(* CoDeSys 2.3.5.6 project: szlendak_02.pro *)
(* Libraries: Standard.lib 31.10.14 11:17:58, SYSLIBCALLBACK.LIB 31.10.14 11:17:58 *)

(* PLC configuration (modules and I/O channels)
Configuration EC4P-200 [Root] node -1, in %IB0 out %QB0 {EC4P_RestartPwrOn = WARMSTART; EC4P_MaxCycleTime = 20; EC4P_Com1BaudRate = 38400; EC4P_CAN1BaudRate = 125KBaud; EC4P_RoutingId = 127; EC4P_EasyNetId = 1; EC4P_EasyNetCfg = 0; EC4P_EasyNetCycleTime = 50; EC4P_RoutingChannel = CAN1; EC4P_IPFlags = 0; EC4P_IPAddress = 0; EC4P_SubNetMask = 0; EC4P_DefaultGateway = 0; EC4P_SummerWinterFlags = 0; EC4P_SummerWinterRule1 = 0; EC4P_SummerWinterRule2 = 0}
  Local I/O [EC4P_LocalIO] node 0, in %IB0 out %QB0 {EC4P_LocalInt = 0}
    I1 AT %IX0.0 [LocalBitInput] Input I1
    I2 AT %IX0.1 [LocalBitInput] Input I2
    I3 AT %IX0.2 [LocalBitInput] Input I3
    I4 AT %IX0.3 [LocalBitInput] Input I4
    I5 AT %IX0.4 [LocalBitInput] Input I5
    I6 AT %IX0.5 [LocalBitInput] Input I6
    I7 AT %IX0.6 [LocalBitInput] Input I7
    I8 AT %IX0.7 [LocalBitInput] Input I8
    I9 AT %IX1.0 [LocalBitInput] Input I9
    I10 AT %IX1.1 [LocalBitInput] Input I10
    I11 AT %IX1.2 [LocalBitInput] Input I11
    I12 AT %IX1.3 [LocalBitInput] Input I12
    I13 AT %IX1.4 [LocalDiagInput] Diagnostic Input I13
    I14 AT %IX1.5 [LocalDiagInput] Diagnostic Input I14
    I15 AT %IX1.6 [LocalDiagInput] Diagnostic Input I15
    I16 AT %IX1.7 [LocalDiagInput] Diagnostic Input I16
    I7_Analog AT %IW2 [LocalAnalogIn] Input I7, 10Bit, 0-10VDC
    I8_Analog AT %IW4 [LocalAnalogIn] Input I8, 10Bit, 0-10VDC
    I11_Analog AT %IW6 [LocalAnalogIn] Input I11, 10Bit, 0-10VDC
    I12_Analog AT %IW8 [LocalAnalogIn] Input I12, 10Bit, 0-10VDC
    Transistor Outputs [EC4P_TOutputs] node 0, in %IB10 out %QB0
      Q1 AT %QX0.0 [LocalBitOutput] Transistor-Output Q1
      Q2 AT %QX0.1 [LocalBitOutput] Transistor-Output Q2
      Q3 AT %QX0.2 [LocalBitOutput] Transistor-Output Q3
      Q4 AT %QX0.3 [LocalBitOutput] Transistor-Output Q4
      Q5 AT %QX0.4 [LocalBitOutput] Transistor-Output Q5
      Q6 AT %QX0.5 [LocalBitOutput] Transistor-Output Q6
      Q7 AT %QX0.6 [LocalBitOutput] Transistor-Output Q7
      Q8 AT %QX0.7 [LocalBitOutput] Transistor-Output Q8
    No Analog Output [EC4P_NoAnalogOutput] node 1, in %IB10 out %QB1
    No Keys [EC4P_NoKeys] node 2, in %IB10 out %QB1
    No Counter [EC4P_NoCounter] node 3, in %IB10 out %QB1
  Extension [EC4P_Extension] node 1, in %IB10 out %QB1
    No Extension [EC4P_NoExtension] node 0, in %IB10 out %QB1
*)

(* Global variable list: Zmienne_globalne *)
VAR_GLOBAL
	K1: BOOL;
	K2: BOOL;
	K3: BOOL;
	f2: BOOL;
	g2: BOOL;
END_VAR

(* POU PLC_PRG, LD *)
PROGRAM PLC_PRG
VAR
	T1: TON;
	T2: TP;
	T4: F_TRIG;
	T3: TP;
	T5: TP;
	T6: F_TRIG;
	T7: TON;
	T8: TP;
	T9: F_TRIG;
	T10: TP;
	T11: F_TRIG;
	T12: TP;
	T13: TP;
	T14: TP;
	T15: TON;
	T16: TP;
	T17: TON;
	x1: BOOL;
	x2: BOOL;
	r1: R_TRIG;
	to1: TOF;
	y1: BOOL;
	r2: F_TRIG;
	to2: TOF;
	y2: BOOL;
	f4: BOOL;
	f3: BOOL;
	f1: BOOL;
	g1: BOOL;
	f6: BOOL;
	f7: BOOL;
	f8: BOOL;
	g3: BOOL;
	g4: BOOL;
END_VAR
VAR_INPUT
	f5: BOOL;
END_VAR
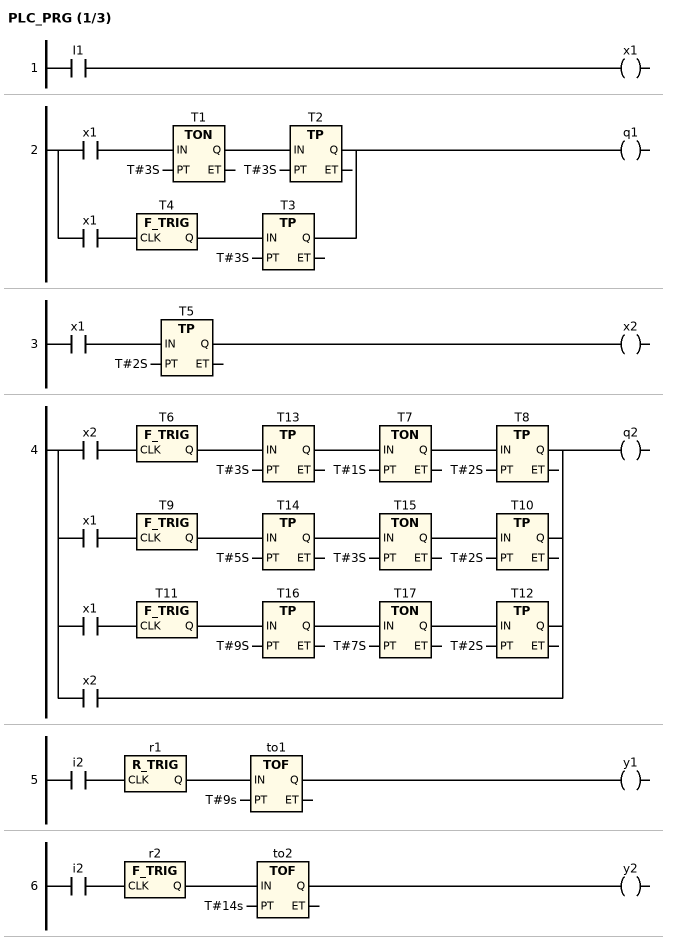
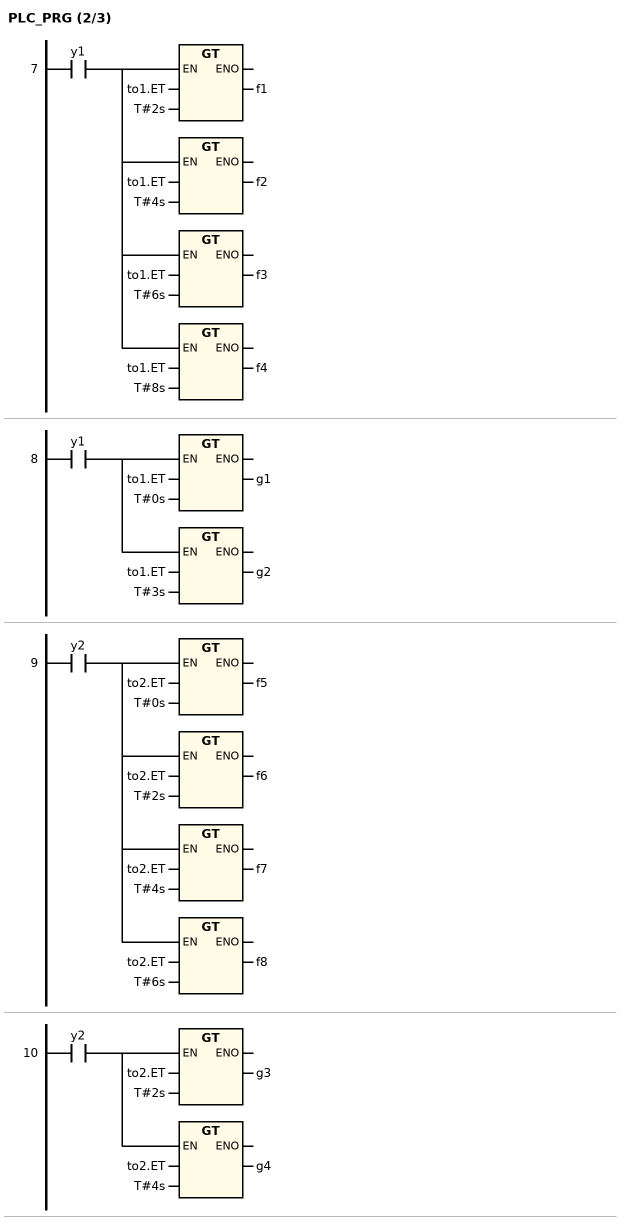
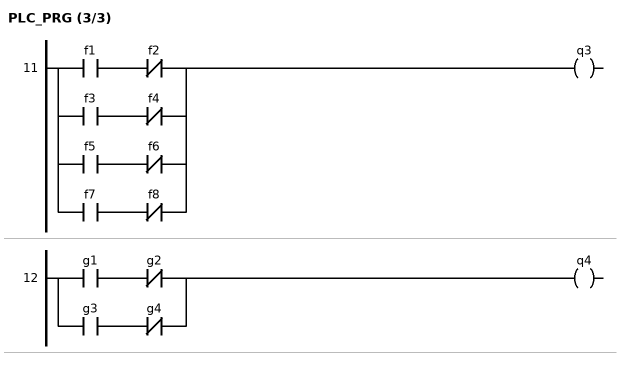
_LD_ (* Ladder Diagram *)
NETWORK 1
	[I1] --- (x1)
NETWORK 2
	{ [x1] - T1:TON(IN: *, PT: T#3S) - T2:TP(IN: *, PT: T#3S) | [x1] - T4:F_TRIG(CLK: *) - T3:TP(IN: *, PT: T#3S) } --- (q1)
NETWORK 3
	[x1] - T5:TP(IN: *, PT: T#2S) --- (x2)
NETWORK 4
	{ [x2] - T6:F_TRIG(CLK: *) - T13:TP(IN: *, PT: T#3S) - T7:TON(IN: *, PT: T#1S) - T8:TP(IN: *, PT: T#2S) | [x1] - T9:F_TRIG(CLK: *) - T14:TP(IN: *, PT: T#5S) - T15:TON(IN: *, PT: T#3S) - T10:TP(IN: *, PT: T#2S) | [x1] - T11:F_TRIG(CLK: *) - T16:TP(IN: *, PT: T#9S) - T17:TON(IN: *, PT: T#7S) - T12:TP(IN: *, PT: T#2S) | [x2] } --- (q2)
NETWORK 5
	[i2] - r1:R_TRIG(CLK: *) - to1:TOF(IN: *, PT: T#9s) --- (y1)
NETWORK 6
	[i2] - r2:F_TRIG(CLK: *) - to2:TOF(IN: *, PT: T#14s) --- (y2)
NETWORK 7
	[y1]
		EN --- GT(to1.ET, T#2s) => f1
		EN --- GT(to1.ET, T#4s) => f2
		EN --- GT(to1.ET, T#6s) => f3
		EN --- GT(to1.ET, T#8s) => f4
NETWORK 8
	[y1]
		EN --- GT(to1.ET, T#0s) => g1
		EN --- GT(to1.ET, T#3s) => g2
NETWORK 9
	[y2]
		EN --- GT(to2.ET, T#0s) => f5
		EN --- GT(to2.ET, T#2s) => f6
		EN --- GT(to2.ET, T#4s) => f7
		EN --- GT(to2.ET, T#6s) => f8
NETWORK 10
	[y2]
		EN --- GT(to2.ET, T#2s) => g3
		EN --- GT(to2.ET, T#4s) => g4
NETWORK 11
	{ [f1] - [/f2] | [f3] - [/f4] | [f5] - [/f6] | [f7] - [/f8] } --- (q3)
NETWORK 12
	{ [g1] - [/g2] | [g3] - [/g4] } --- (q4)
_END_LD_
(* the same logic as Structured Text *)
(* Network 1 *)
x1 := I1;
(* Network 2 *)
T1(IN := x1, PT := T#3S);
T2(IN := T1.Q, PT := T#3S);
T4(CLK := x1);
T3(IN := T4.Q, PT := T#3S);
q1 := T2.Q OR T3.Q;
(* Network 3 *)
T5(IN := x1, PT := T#2S);
x2 := T5.Q;
(* Network 4 *)
T6(CLK := x2);
T13(IN := T6.Q, PT := T#3S);
T7(IN := T13.Q, PT := T#1S);
T8(IN := T7.Q, PT := T#2S);
T9(CLK := x1);
T14(IN := T9.Q, PT := T#5S);
T15(IN := T14.Q, PT := T#3S);
T10(IN := T15.Q, PT := T#2S);
T11(CLK := x1);
T16(IN := T11.Q, PT := T#9S);
T17(IN := T16.Q, PT := T#7S);
T12(IN := T17.Q, PT := T#2S);
q2 := T8.Q OR T10.Q OR T12.Q OR x2;
(* Network 5 *)
r1(CLK := i2);
to1(IN := r1.Q, PT := T#9s);
y1 := to1.Q;
(* Network 6 *)
r2(CLK := i2);
to2(IN := r2.Q, PT := T#14s);
y2 := to2.Q;
(* Network 7 *)
IF y1 THEN
	f1 := to1.ET > T#2s;
	f2 := to1.ET > T#4s;
	f3 := to1.ET > T#6s;
	f4 := to1.ET > T#8s;
END_IF;
(* Network 8 *)
IF y1 THEN
	g1 := to1.ET > T#0s;
	g2 := to1.ET > T#3s;
END_IF;
(* Network 9 *)
IF y2 THEN
	f5 := to2.ET > T#0s;
	f6 := to2.ET > T#2s;
	f7 := to2.ET > T#4s;
	f8 := to2.ET > T#6s;
END_IF;
(* Network 10 *)
IF y2 THEN
	g3 := to2.ET > T#2s;
	g4 := to2.ET > T#4s;
END_IF;
(* Network 11 *)
q3 := f1 AND NOT f2 OR f3 AND NOT f4 OR f5 AND NOT f6 OR f7 AND NOT f8;
(* Network 12 *)
q4 := g1 AND NOT g2 OR g3 AND NOT g4;
END_PROGRAM
